FUNCTION_BLOCK AI_SCALE (* Scale Analog Input Value to Engineering Units *)
  (* Standard: 61499-1; Function: Scaling *)
  (* Version 0.0, 2005-02-22, JHC, Rockwell Automation *)
  (* Compiler header: package fb.rt.process; *)
  (* Compiler Java Sun JDK 1.4.2 *)
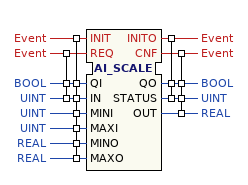
  EVENT_INPUT
    INIT WITH IN, MINI, MAXI, MINO, MAXO, QI; (* Initialization Request *)
    REQ WITH IN, QI; (* Normal Execution Request *)
  END_EVENT
  EVENT_OUTPUT
    INITO WITH QO, STATUS; (* Initialization Confirm *)
    CNF WITH QO, STATUS, OUT; (* Execution Confirmation *)
  END_EVENT
  VAR_INPUT
    QI : BOOL; (* Event Input Qualifier *)
    IN : UINT; (* Analog input measurement *)
    MINI : UINT; (* Minimum IN value *)
    MAXI : UINT := 1024; (* Maximum IN value *)
    MINO : REAL; (* OUT value corresponding to MINI *)
    MAXO : REAL := 1.0; (* OUT value corresponding to MAXI *)
  END_VAR
  VAR_OUTPUT
    QO : BOOL; (* Output event qualifier *)
    STATUS : UINT; (* 0=OK, 1=Inhibited, 2=Bad Scale Factor, 3=Out of Range *)
    OUT : REAL; (* IN scaled to Engineering Units *)
  END_VAR
  VAR
    SF_OK : BOOL; (* SF value is valid *)
    SF : REAL; (* Scale Factor *)
  END_VAR
  ALGORITHM INIT IN Java: (* Initialization algorithm *)
QO.value = QI.value;
STATUS.value = 0;
if(QO.value){
  SF.value = MAXI.value - MINI.value;
  SF_OK.value = (SF.value != 0.0);
  QO.value = SF_OK.value;
  if(QO.value) SF.value = (MAXO.value-MINO.value)/SF.value;
  else STATUS.value = 2;}
else SF_OK.value = false;
INITO.serviceEvent(this);
  END_ALGORITHM
  ALGORITHM REQ IN Java: (* Normally executed algorithm *)
QO.value = QI.value;
STATUS.value = 0;
if(!QO.value) STATUS.value=1;
else if(!SF_OK.value){
   QO.value = false;
   STATUS.value=2;}
else if(IN.value<MINI.value){
   QO.value = false;
   STATUS.value = 3;
   OUT.value = MINO.value;}
else if(IN.value>MAXI.value){
   QO.value = false;
   STATUS.value = 3;
   OUT.value = MAXO.value;}
else OUT.value = MINO.value+(IN.value-MINI.value)*SF.value;
CNF.serviceEvent(this);
  END_ALGORITHM
END_FUNCTION_BLOCK
